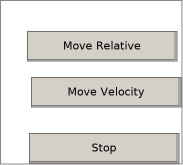
VISUALIZATION Vis_Axis  // 183x165
    Button (27,31 150x30), "Move Relative"
        tap gHMI.bMoveRel
    Button (31,77 150x30), "Move Velocity"
        tap gHMI.bMoveVel
    Button (29,133 150x30), "Stop"
        tap gHMI.bStop
END_VISUALIZATION

(* stored: Version 1.1.0.1, ProductVersion 3.1.4024.0
   Visu Vis_Axis: Id {3f34c172-c1f1-4f7a-ba0c-083ec4acc86b} *)
